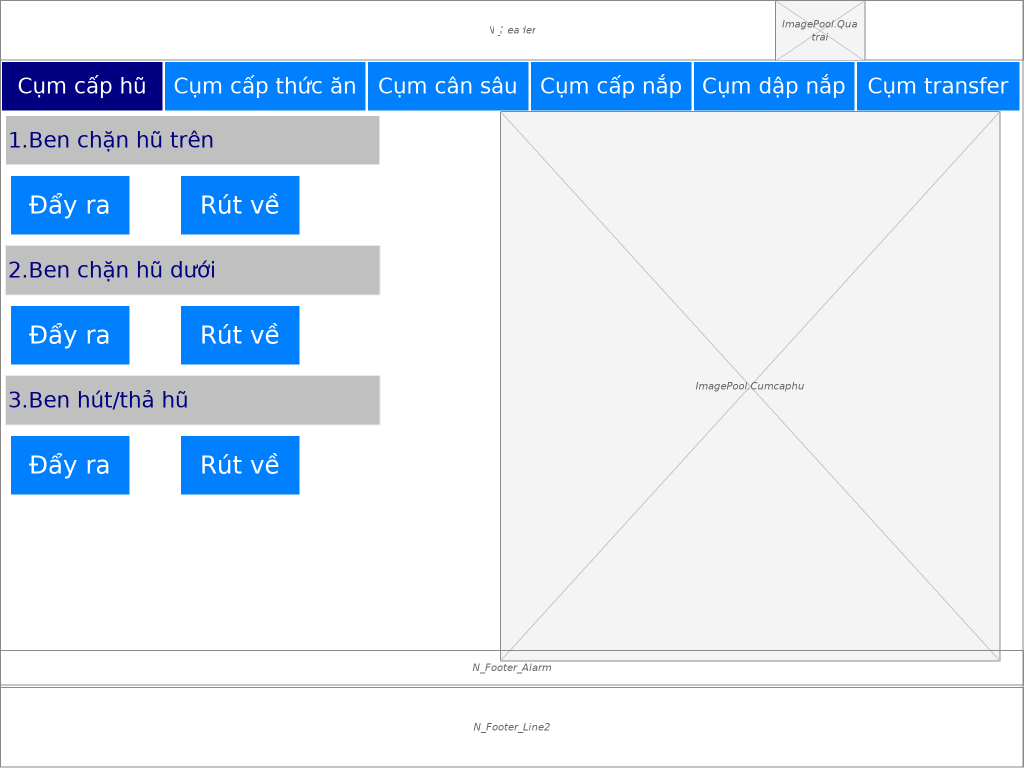
VISUALIZATION N_JarSupply2  // 1024x768
    Rectangle (10,305 120x60), "Đẩy ra", colour toggle: PR_Line02.bCylinder_dw_extend
        OnMouseDown: execute { PR_Line02.bCylinder_dw_extend := TRUE; PR_Line02.bCylinder_dw_retract := FALSE; }
    Rectangle (180,175 120x60), "Rút về", colour toggle: PR_Line02.bCylinder_up_retract
        OnMouseDown: execute { PR_Line02.bCylinder_up_retract := TRUE; PR_Line02.bCylinder_up_extend := FALSE; }
    Rectangle (180,305 120x60), "Rút về", colour toggle: PR_Line02.bCylinder_dw_retract
        OnMouseDown: execute { PR_Line02.bCylinder_dw_retract := TRUE; PR_Line02.bCylinder_dw_extend := FALSE; }
    Frame (0,687 1024x80)
        shows N_Footer_Line2()
    Frame (0,0 1024x60)
        shows N_Header()
    Textfield (353,5 400x50), "MÀN HÌNH CHẠY TAY LINE 2"
    Rectangle (10,175 120x60), "Đẩy ra", colour toggle: PR_Line02.bCylinder_up_extend
        OnMouseDown: execute { PR_Line02.bCylinder_up_extend := TRUE; PR_Line02.bCylinder_up_retract := FALSE; }
    Image (775,0 90x61), input disabled if: bResetAuto1, image: ImagePool.Qua trai
        OnMouseClick: change screen: N_JarSupply1
        OnMouseClick: execute { MAIN.bModeManual := TRUE; MAIN.bModeAuto := FALSE; }
    Rectangle (1,61 162x50), "Cụm cấp hũ"
        OnMouseClick: change screen: N_JarSupply2
    Rectangle (164,61 202x50), "Cụm cấp thức ăn"
        OnMouseClick: change screen: N_FoodSupply2
    Rectangle (367,61 162x50), "Cụm cân sâu"
        OnMouseClick: change screen: N_WormWeight2
    Rectangle (530,61 162x50), "Cụm cấp nắp"
        OnMouseClick: change screen: N_LidSupply2
    Rectangle (693,61 162x50), "Cụm dập nắp"
        OnMouseClick: change screen: N_LidPressing2
    Rectangle (856,61 164x50), "Cụm transfer"
        OnMouseClick: change screen: N_Tranfer2
    Rectangle (5,115 375x50), "1.Ben chặn hũ trên"
    Rectangle (5,245 375x50), "2.Ben chặn hũ dưới"
    Image (500,111 500x550), image: ImagePool.Cumcaphu
    Frame (0,650 1024x35)
        shows N_Footer_Alarm()
    Rectangle (10,435 120x60), "Đẩy ra", colour toggle: PR_Line02.bCylinder_Suction_cup_extend
        OnMouseDown: execute { PR_Line02.bCylinder_Suction_cup_extend := TRUE; PR_Line02.bCylinder_Suction_cup_retract := FALSE; }
    Rectangle (180,435 120x60), "Rút về", colour toggle: PR_Line02.bCylinder_Suction_cup_retract
        OnMouseDown: execute { PR_Line02.bCylinder_Suction_cup_extend := FALSE; PR_Line02.bCylinder_Suction_cup_retract := true; }
    Rectangle (5,375 375x50), "3.Ben hút/thả hũ"
END_VISUALIZATION

(* stored: Version 1.1.0.1, ProductVersion 3.1.4024.12
   Visu N_JarSupply2: Id {101b5048-ebea-46d4-9179-59d644674010} *)
